Omron CX-Programmer project NewProject (CX-Programmer 9.51)

# PLC NewPLC1: CP1L L
; My_First_Project

## Program NewProgram1 (cyclic task 0)
Local symbols
button_1 0.00 BOOL  ; COMMENT
out_1 100.01 BOOL
out_2 100.01 BOOL

### Section Section1

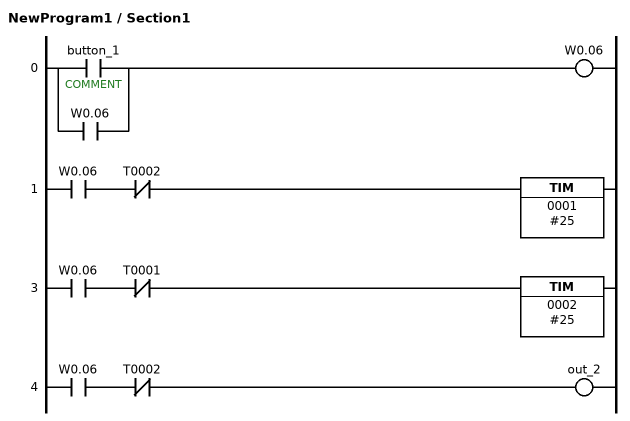
; rung 0
LD button_1  ; COMMENT
OR W0.06
OUT W0.06
; rung 1
LD W0.06
ANDNOT T0002
TIM 0001 #25
; rung 3
LD W0.06
ANDNOT T0001
TIM 0002 #25
; rung 4
LD W0.06
ANDNOT T0002
OUT out_2

### Section END
; rung 0
END(001)